Staubli VAL3: find.pgx

public program find(string& x_sItem[], bool& x_bFound[])
  local num i
  local num l_nSize
  local string l_sItem
begin
  // find an item in the list
  x_bFound=isDefined(saveInOut:dInput[x_sItem])
end
